// TIA Portal V21 export
VAR_GLOBAL   // PLC tag table "INSTRUMENTOS (ETA)"
   "FIT-01_STS" AT %M61.0 : Bool;
   "LIT-01_STS" AT %M61.1 : Bool;
END_VAR
